TYPE Case_step :
STRUCT
END_STRUCT
END_TYPE

(* stored: Version 1.1.0.1, ProductVersion 3.1.4024.15
   DUT Case_step: Id {c70091eb-cf00-466f-ae3f-fb86165ace4b} *)
